VAR_GLOBAL
	
	// ================================================================
    // RAIL 1
    // ================================================================
	R1_Sensor_UnknownState : ST_Alarm := (
		nID := 1001,
		nSeverity := 3);
	
	R1_Sensor_MotionTimedOut : ST_Alarm := (
		nID := 1002,
		nSeverity := 3);
	
	R1_Chariot_UnknownState : ST_Alarm := (
		nID := 1003,
		nSeverity := 3);
	
	R1_Chariot_MotionTimedOut : ST_Alarm := (
		nID := 1004,
		nSeverity := 3);
	
	R1_Compressor_UnknownState : ST_Alarm := (
		nID := 1005,
		nSeverity := 3);
	
	R1_Compressor_MotionTimedOut : ST_Alarm := (
		nID := 1006,
		nSeverity := 3);
	
	R1_Stepper_Motion_Failed : ST_Alarm := (
		sMessage := '',
		nID := 1007,
		nSeverity := 3);
	
	R1_Stepper_Homing_Failed : ST_Alarm := (
		sMessage := '',
		nID := 1008,
		nSeverity := 3);
	
	R1_Stepper_Motion_Interrupted : ST_Alarm := (
		sMessage := '',
		nID := 1010,
		nSeverity := 3);
	
	R1_Stepper_PowerUp_Failed : ST_Alarm := (
		sMessage := '',
		nID := 1011,
		nSeverity := 3);
	
	R1_Stepper_Reset_Failed : ST_Alarm := (
		sMessage := '',
		nID := 1012,
		nSeverity := 3);
	
	R1_Stepper_Stop_Failed : ST_Alarm := (
		sMessage := '',
		nID := 1013,
		nSeverity := 3);
	
	R1_Stepper_UnableToReadPosition : ST_Alarm := (
		sMessage := '',
		nID := 1014,
		nSeverity := 3);
	
	R1_Compressor_DriveFaulted : ST_Alarm := (
		nID := 1015,
		nSeverity := 5);
	
	
	// ================================================================
    // RAIL 2
    // ================================================================
	R2_Stepper_PowerUp_Failed : ST_Alarm := (
		sMessage := '',
		nID := 2001,
		nSeverity := 3);
	
	R2_Stepper_Homing_Failed : ST_Alarm := (
		sMessage := '',
		nID := 2002,
		nSeverity := 3);
	
	R2_Stepper_Motion_Failed : ST_Alarm := (
		sMessage := '',
		nID := 2004,
		nSeverity := 3);
	
	R2_Stepper_Motion_Interrupted : ST_Alarm := (
		sMessage := '',
		nID := 2005,
		nSeverity := 3);
	
	R2_Stepper_Reset_Failed : ST_Alarm := (
		sMessage := '',
		nID := 2006,
		nSeverity := 3);
		
	R2_Chariot_UnknownState : ST_Alarm := (
		nID := 2007,
		nSeverity := 3);
	
	R2_Chariot_MotionTimedOut : ST_Alarm := (
		nID := 2008,
		nSeverity := 3);
	
	R2_Stepper_Stop_Failed : ST_Alarm := (
		sMessage := '',
		nID := 2009,
		nSeverity := 3);
	
	R2_Stepper_UnableToReadPosition : ST_Alarm := (
		sMessage := '',
		nID := 2010,
		nSeverity := 3);
	
	
	// ================================================================
    // RAIL 3
    // ================================================================
	R3_Compressor_UnknownState : ST_Alarm := (
		nID := 3001,
		nSeverity := 3);
	
	R3_Compressor_MotionTimedOut : ST_Alarm := (
		nID := 3002,
		nSeverity := 3);
	
	R3_HeatExCoupola_UnknownState : ST_Alarm := (
		nID := 3003,
		nSeverity := 3);
	
	R3_HeatExCoupola_MotionTimedOut : ST_Alarm := (
		nID := 3004,
		nSeverity := 3);
	
	R3_RegenCoupola_UnknownState : ST_Alarm := (
		nID := 3005,
		nSeverity := 3);
	
	R3_RegenCoupola_MotionTimedOut : ST_Alarm := (
		nID := 3006,
		nSeverity := 3);
	
	R3_Chariot_UnknownState : ST_Alarm := (
		nID := 3007,
		nSeverity := 3);
	
	R3_Chariot_MotionTimedOut : ST_Alarm := (
		nID := 3008,
		nSeverity := 3);
		
	R3_Stepper_PowerUp_Failed : ST_Alarm := (
		sMessage := '',
		nID := 3009,
		nSeverity := 3);
	
	R3_Stepper_Homing_Failed : ST_Alarm := (
		sMessage := '',
		nID := 3010,
		nSeverity := 3);
	
	R3_Stepper_Motion_Failed : ST_Alarm := (
		sMessage := '',
		nID := 3012,
		nSeverity := 3);
	
	R3_Stepper_Motion_Interrupted : ST_Alarm := (
		sMessage := '',
		nID := 3013,
		nSeverity := 3);
	
	R3_Stepper_Reset_Failed : ST_Alarm := (
		sMessage := '',
		nID := 3014,
		nSeverity := 3);
	
	R3_Stepper_Stop_Failed : ST_Alarm := (
		sMessage := '',
		nID := 3015,
		nSeverity := 3);
	
	R3_HeatExCoupola_DriveFaulted : ST_Alarm := (
		nID := 3016,
		nSeverity := 5);
	
	R3_RegenCoupola_DriveFaulted : ST_Alarm := (
		nID := 3017,
		nSeverity := 5);
	
	R3_Stepper_UnableToReadPosition : ST_Alarm := (
		sMessage := '',
		nID := 3018,
		nSeverity := 3);
	
	R3_Compressor_DriveFaulted : ST_Alarm := (
		nID := 3019,
		nSeverity := 5);
	
	// ================================================================
    // RAIL 4
    // ================================================================
	R4_Stepper_PowerUp_Failed : ST_Alarm := (
		sMessage := '',
		nID := 4001,
		nSeverity := 3);
	
	R4_Stepper_Homing_Failed : ST_Alarm := (
		sMessage := '',
		nID := 4002,
		nSeverity := 3);
	
	R4_Stepper_Motion_Failed : ST_Alarm := (
		sMessage := '',
		nID := 4004,
		nSeverity := 3);
	
	R4_Stepper_Motion_Interrupted : ST_Alarm := (
		sMessage := '',
		nID := 4005,
		nSeverity := 3);
	
	R4_Stepper_Reset_Failed : ST_Alarm := (
		sMessage := '',
		nID := 4006,
		nSeverity := 3);
	
	R4_Chariot_UnknownState : ST_Alarm := (
		nID := 4007,
		nSeverity := 3);
	
	R4_Chariot_MotionTimedOut : ST_Alarm := (
		nID := 4008,
		nSeverity := 3);
	
	R4_Stepper_Stop_Failed : ST_Alarm := (
		sMessage := '',
		nID := 4009,
		nSeverity := 3);
	
	R4_Stepper_UnableToReadPosition : ST_Alarm := (
		sMessage := '',
		nID := 4010,
		nSeverity := 3);
	
	
	// ================================================================
    // GLOBAL SECURITY (ZONE 5)
    // ================================================================
	SafetyRelay : ST_Alarm := (
		nID := 9001,
		nSeverity := 5);
	
	bCriticalAlarm : BOOL;
END_VAR

(* stored: Version 1.1.0.1, ProductVersion 3.1.4026.11
   GVL GVL_Alarms: Id {637d89bc-47d1-47bf-b0f7-7f6be8b20113} *)
